FUNCTION_BLOCK FB_ReceiveabcCurrent_Left
VAR_IN_OUT
	Inputs_Left : CANRXQUEUESTRUCT_E_32;
	Outputs_Left : CANTXQUEUESTRUCT_E_32;
END_VAR
VAR_OUTPUT
	Ia_Left : LREAL;
	Ib_Left : LREAL;
	Ic_Left : LREAL;
END_VAR
VAR
	MessageReceived : ARRAY[0..31] OF EXTCANQUEUE;
	i : INT;
	fbPPS_Timer : TON;
	nPacketsPerSecond: INT;
	nReceiveCounter : INT;
	nLastReceiveCounter : INT;
	
END_VAR

FOR i := 0 TO (Inputs_Left.NoOfRxMessages-1) DO
    IF Inputs_Left.RxMessages[i].cobId = 600 THEN 
        Ia_Left := INT_TO_LREAL(WORD_TO_INT(SHL(USINT_TO_UINT(Inputs_Left.RxMessages[i].data[0]), 8) OR USINT_TO_UINT(Inputs_Left.RxMessages[i].data[1]))) / 10.0; 
        Ib_Left := INT_TO_LREAL(WORD_TO_INT(SHL(USINT_TO_UINT(Inputs_Left.RxMessages[i].data[2]), 8) OR USINT_TO_UINT(Inputs_Left.RxMessages[i].data[3]))) / 10.0; 
        Ic_Left := INT_TO_LREAL(WORD_TO_INT(SHL(USINT_TO_UINT(Inputs_Left.RxMessages[i].data[4]), 8) OR USINT_TO_UINT(Inputs_Left.RxMessages[i].data[5]))) / 10.0;
		
		nReceiveCounter := nReceiveCounter + 1;
    END_IF
END_FOR
fbPPS_Timer(IN := NOT fbPPS_Timer.Q, PT := T#1S);
IF fbPPS_Timer.Q THEN
			nPacketsPerSecond   := nReceiveCounter - nLastReceiveCounter;
			nLastReceiveCounter := nReceiveCounter;
END_IF

END_FUNCTION_BLOCK

(* stored: Version 1.1.0.1
   POU FB_ReceiveabcCurrent_Left: Id {d0e9e005-20e4-40bb-8e0b-987459c2a14d}, SpecialFunc None *)
